// TIA Portal V18 export
FUNCTION "ACC_Main" : Void   // FC6, LAD
{ S7_Optimized_Access := 'TRUE' }
VERSION : 0.1
// stored: AutoNumber true, IsIECCheckEnabled false, SetENOAutomatically false, UDAEnableTagReadback false
BEGIN

REGION Network 1: 区域搜索
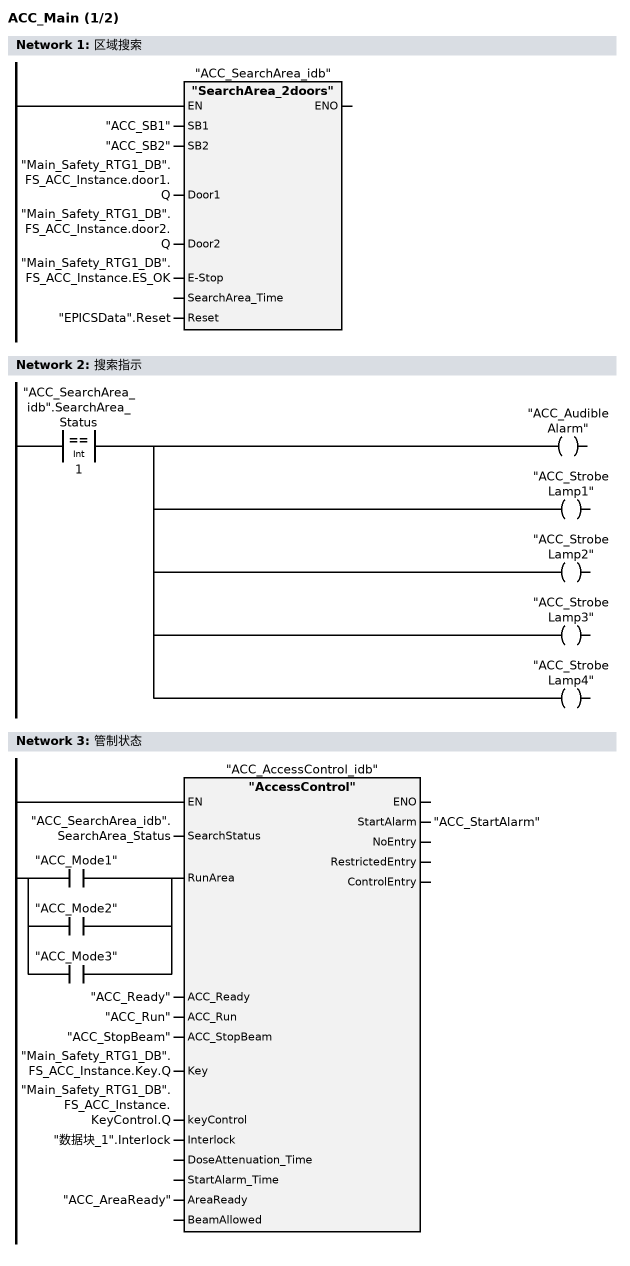
   RUNG wire#powerrail
      "ACC_SearchArea_idb"(SB1 := "ACC_SB1", SB2 := "ACC_SB2", Door1 := "Main_Safety_RTG1_DB".FS_ACC_Instance.door1.Q, Door2 := "Main_Safety_RTG1_DB".FS_ACC_Instance.door2.Q, "E-Stop" := "Main_Safety_RTG1_DB".FS_ACC_Instance.ES_OK, SearchArea_Time :=, Reset := "EPICSData".Reset)
   END_RUNG
   // the same network as SCL:
   "ACC_SearchArea_idb"(SB1 := "ACC_SB1",   // "SearchArea_2doors"
                        SB2 := "ACC_SB2",
                        Door1 := "Main_Safety_RTG1_DB".FS_ACC_Instance.door1.Q,
                        Door2 := "Main_Safety_RTG1_DB".FS_ACC_Instance.door2.Q,
                        "E-Stop" := "Main_Safety_RTG1_DB".FS_ACC_Instance.ES_OK,
                        Reset := "EPICSData".Reset);
END_REGION

REGION Network 2: 搜索指示
   RUNG wire#powerrail
      { S7_Templates := "SrcType := Int" } EQ_Contact(in1 := "ACC_SearchArea_idb".SearchArea_Status, in2 := 1)
      wire#w1
      Coil( "ACC_AudibleAlarm" )
   END_RUNG
   RUNG wire#w1
      Coil( "ACC_StrobeLamp1" )
   END_RUNG
   RUNG wire#w1
      Coil( "ACC_StrobeLamp2" )
   END_RUNG
   RUNG wire#w1
      Coil( "ACC_StrobeLamp3" )
   END_RUNG
   RUNG wire#w1
      Coil( "ACC_StrobeLamp4" )
   END_RUNG
   // the same network as SCL:
   "ACC_AudibleAlarm" := "ACC_SearchArea_idb".SearchArea_Status = 1;
   "ACC_StrobeLamp1" := "ACC_AudibleAlarm";
   "ACC_StrobeLamp2" := "ACC_AudibleAlarm";
   "ACC_StrobeLamp3" := "ACC_AudibleAlarm";
   "ACC_StrobeLamp4" := "ACC_AudibleAlarm";
END_REGION

REGION Network 3: 管制状态
   RUNG wire#powerrail
      "ACC_AccessControl_idb"(RunArea := wire#w1, SearchStatus := "ACC_SearchArea_idb".SearchArea_Status, ACC_Ready := "ACC_Ready", ACC_Run := "ACC_Run", ACC_StopBeam := "ACC_StopBeam", Key := "Main_Safety_RTG1_DB".FS_ACC_Instance.Key.Q, keyControl := "Main_Safety_RTG1_DB".FS_ACC_Instance.KeyControl.Q, Interlock := "数据块_1".Interlock, DoseAttenuation_Time :=, StartAlarm_Time :=, AreaReady := "ACC_AreaReady", BeamAllowed :=, StartAlarm => "ACC_StartAlarm", NoEntry =>, RestrictedEntry =>, ControlEntry =>)
   END_RUNG
   RUNG wire#powerrail
      Contact( "ACC_Mode1" )
   END_RUNG wire#w1
   RUNG wire#powerrail
      Contact( "ACC_Mode2" )
   END_RUNG wire#w1
   RUNG wire#powerrail
      Contact( "ACC_Mode3" )
   END_RUNG wire#w1
   // the same network as SCL:
   "ACC_AccessControl_idb"(SearchStatus := "ACC_SearchArea_idb".SearchArea_Status,   // "AccessControl"
                           RunArea := "ACC_Mode1" OR "ACC_Mode2" OR "ACC_Mode3",
                           ACC_Ready := "ACC_Ready",
                           ACC_Run := "ACC_Run",
                           ACC_StopBeam := "ACC_StopBeam",
                           Key := "Main_Safety_RTG1_DB".FS_ACC_Instance.Key.Q,
                           keyControl := "Main_Safety_RTG1_DB".FS_ACC_Instance.KeyControl.Q,
                           Interlock := "数据块_1".Interlock,
                           AreaReady := "ACC_AreaReady",
                           StartAlarm => "ACC_StartAlarm");
END_REGION

REGION Network 4: 管制输出
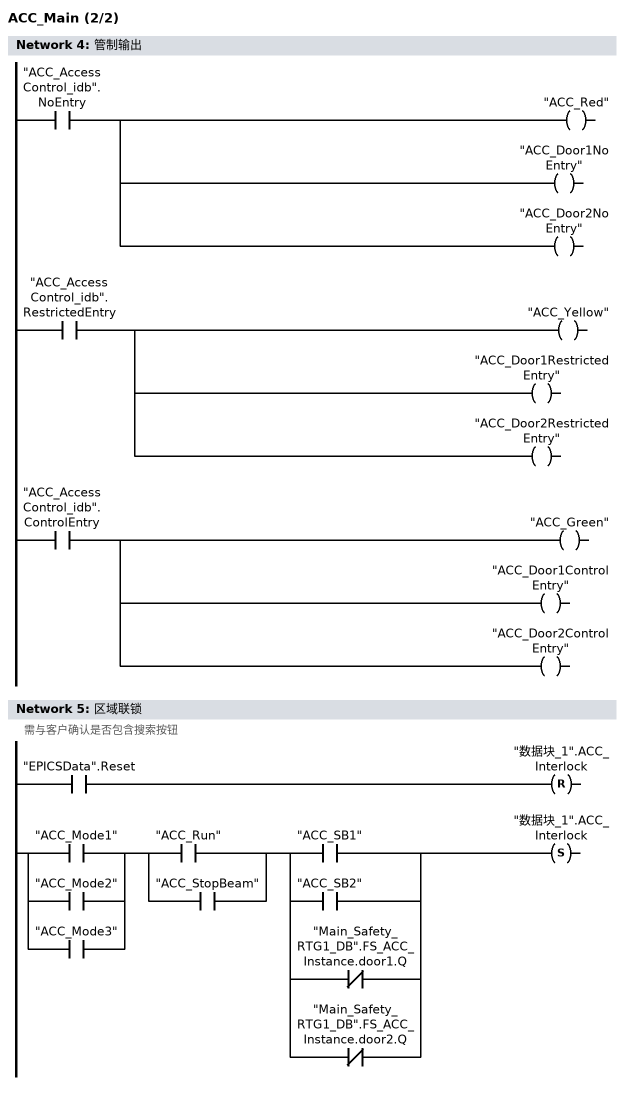
   RUNG wire#powerrail
      Contact( "ACC_AccessControl_idb".NoEntry )
      wire#w1
      Coil( "ACC_Red" )
   END_RUNG
   RUNG wire#w1
      Coil( "ACC_Door1NoEntry" )
   END_RUNG
   RUNG wire#w1
      Coil( "ACC_Door2NoEntry" )
   END_RUNG
   RUNG wire#powerrail
      Contact( "ACC_AccessControl_idb".RestrictedEntry )
      wire#w2
      Coil( "ACC_Yellow" )
   END_RUNG
   RUNG wire#w2
      Coil( "ACC_Door1RestrictedEntry" )
   END_RUNG
   RUNG wire#w2
      Coil( "ACC_Door2RestrictedEntry" )
   END_RUNG
   RUNG wire#powerrail
      Contact( "ACC_AccessControl_idb".ControlEntry )
      wire#w3
      Coil( "ACC_Green" )
   END_RUNG
   RUNG wire#w3
      Coil( "ACC_Door1ControlEntry" )
   END_RUNG
   RUNG wire#w3
      Coil( "ACC_Door2ControlEntry" )
   END_RUNG
   // the same network as SCL:
   "ACC_Red" := "ACC_AccessControl_idb".NoEntry;
   "ACC_Door1NoEntry" := "ACC_AccessControl_idb".NoEntry;
   "ACC_Door2NoEntry" := "ACC_AccessControl_idb".NoEntry;
   "ACC_Yellow" := "ACC_AccessControl_idb".RestrictedEntry;
   "ACC_Door1RestrictedEntry" := "ACC_AccessControl_idb".RestrictedEntry;
   "ACC_Door2RestrictedEntry" := "ACC_AccessControl_idb".RestrictedEntry;
   "ACC_Green" := "ACC_AccessControl_idb".ControlEntry;
   "ACC_Door1ControlEntry" := "ACC_AccessControl_idb".ControlEntry;
   "ACC_Door2ControlEntry" := "ACC_AccessControl_idb".ControlEntry;
END_REGION

REGION Network 5: 区域联锁
   // 需与客户确认是否包含搜索按钮
   RUNG wire#powerrail
      Contact( "EPICSData".Reset )
      R_Coil( "数据块_1".ACC_Interlock )
   END_RUNG
   RUNG wire#powerrail
      Contact( "ACC_Mode1" )
      wire#w1
      Contact( "ACC_Run" )
      wire#w2
      Contact( "ACC_SB1" )
      wire#w3
      S_Coil( "数据块_1".ACC_Interlock )
   END_RUNG
   RUNG wire#powerrail
      Contact( "ACC_Mode2" )
   END_RUNG wire#w1
   RUNG wire#powerrail
      Contact( "ACC_Mode3" )
   END_RUNG wire#w1
   RUNG wire#w1
      Contact( "ACC_StopBeam" )
   END_RUNG wire#w2
   RUNG wire#w2
      Contact( "ACC_SB2" )
   END_RUNG wire#w3
   RUNG wire#w2
      I_Contact( "Main_Safety_RTG1_DB".FS_ACC_Instance.door1.Q )
   END_RUNG wire#w3
   RUNG wire#w2
      I_Contact( "Main_Safety_RTG1_DB".FS_ACC_Instance.door2.Q )
   END_RUNG wire#w3
   // the same network as SCL:
   IF "EPICSData".Reset THEN "数据块_1".ACC_Interlock := FALSE; END_IF;
   IF ("ACC_Mode1" OR "ACC_Mode2" OR "ACC_Mode3") AND ("ACC_Run" OR "ACC_StopBeam") AND ("ACC_SB1" OR "ACC_SB2" OR NOT "Main_Safety_RTG1_DB".FS_ACC_Instance.door1.Q OR NOT "Main_Safety_RTG1_DB".FS_ACC_Instance.door2.Q) THEN
       "数据块_1".ACC_Interlock := TRUE;
   END_IF;
END_REGION
END_FUNCTION
